# EPICS autosave request: tests/testfiles/cfg/SF_BPM_PV.req
$(SYS):X-OFFS
$(SYS):Y-OFFS
$(SYS):T1-OFFS
$(SYS):T2-OFFS
$(SYS):X-REF-FB
$(SYS):Y-REF-FB
